# EPICS substitutions: evrSupport/Db/ioc/bsaXL01.substitutions
#####################
# BSA functionality for devices
# load these for sim or real data
####################
file bsaBPMSEdef.template {
  pattern {DEVICE  , IOCI , EVRI}
	  { BPMS:XX01:1, SYS0 , IOC:XX01:1}
	  { BPMS:XX01:2, SYS0 , IOC:XX01:1}
	  { BPMS:XX01:3, SYS0 , IOC:XX01:1}
	  { BPMS:XX01:4, SYS0 , IOC:XX01:1}
	  { BPMS:XX01:5, SYS0 , IOC:XX01:1}
	  { BPMS:XX01:6, SYS0 , IOC:XX01:1}
}

file bsaTOROEdef.template {
  pattern {DEVICE   , IOCI , EVRI}
	  { TORO:XX01:1 , SYS0 , IOC:XX01:1}
	  { TORO:XX01:2 , SYS0 , IOC:XX01:1}
}
file bsaPMTEdef.template {
  pattern { DEVICE , IOCI , EVRI }
	  { PMT:XX01:1 , SYS0 , IOC:XX01:1}
	  { PMT:XX01:2 , SYS0 , IOC:XX01:1}
	  { PMT:XX01:3 , SYS0 , IOC:XX01:1}
	  { PMT:XX01:4 , SYS0 , IOC:XX01:1}
	  { PMT:XX01:5 , SYS0 , IOC:XX01:1}
	  { PMT:XX01:6 , SYS0 , IOC:XX01:1}
}
file bsaBLENEdef.template {
  pattern { DEVICE ,  IOCI, EVRI }
	  { BLEN:XX01:1 , SYS0, IOC:XX01:1 }
	  { BLEN:XX01:2 , SYS0, IOC:XX01:1 }
	  { BLEN:XX01:3 , SYS0, IOC:XX01:1 }
}
file bsaKICKEdef.template {
  pattern { DEVICE  , IOCI , EVRI}
	  { KICK:XX01:1 , SYS0 , IOC:XX01:1}
	  { KICK:XX01:2 , SYS0 , IOC:XX01:1}
	  { KICK:XX01:3 , SYS0 , IOC:XX01:1}
}
file bsaWIREEdef.template {
  pattern { DEVICE  , IOCI , EVRI}
	  { WIRE:XX01:1 , SYS0 , IOC:XX01:1}
	  { WIRE:XX01:2 , SYS0 , IOC:XX01:1}
	  { WIRE:XX01:3 , SYS0 , IOC:XX01:1}
	  { WIRE:XX01:4 , SYS0 , IOC:XX01:1}
}
#
# Pattern records
file evrPattern.template {
#	    Device    ,  SLC Pattern Check LNK     ,  EVR/Trigger          Diagnostic
#	                                                 Links                Link
  pattern { DEVICE     ,        LINK4              , LINK5 ,   LINK6    ,          LINKD      }
	  { IOC:XX01:1 , "IOC:XX01:1:FANOUTSLC PP" ,  ""   ,    ""      , "IOC:XX01:1:YYD PP" }
}
file evrPatternProc.template {
  pattern { DEVICE }
	  { IOC:XX01:1}
}
